TYPE ST_DigitalInputOutCmd :
STRUCT
    Reserved : BOOL; // passive monitor: no command result
END_STRUCT
END_TYPE

(* stored: Version 1.1.0.1, ProductVersion 3.1.4024.12
   DUT ST_DigitalInputOutCmd: Id {f622c5b7-4b4d-4c6a-a722-23d353a5a4b8} *)
